// TIA Portal V16 export
// export: Created 2023-03-29T11:03:44.8927615Z, ExportSetting WithDefaults, DisplayName Totally Integrated Automation Portal, DisplayVersion V16 Update 6, DisplayName TIA Portal Version Control Interface, DisplayVersion V16 Update 2, DisplayName TIA Portal Openness, DisplayVersion V16 Update 6, DisplayName STEP 7 Professional, DisplayVersion V16 Update 6, DisplayName STEP 7 Safety, DisplayVersion V16, DisplayName WinCC Advanced, DisplayVersion V16 Update 6
VAR_GLOBAL   // PLC tag table "Z3"
   Hbit_Alarm_Z3 AT %M14.0 : Bool;
   CMD_Open_Z_3 AT %M57.5 : Bool;   // załącz otwieranie
   Hbit_Reset_Z3 AT %M14.6 : Bool;
   CMD_Awaria_Z_3 AT %M57.7 : Bool;   // Awaria zbiorcza
   inputOtwartaZ_3 AT %M56.2 : Bool;   // znacznik wejście
   setAlarm_Moment_Z_3 AT %M57.4 : Bool;   // znacznik alarmu od momentówki w trybie zdalnym (aut/mamnual)
   inputRuch_Z_3 AT %M56.4 : Bool;
   setSVMO_Z_3 AT %M57.2 : Bool;   // Znacznik polecenia otwórz w trybie automat
   CMD_Close_Z_3 AT %M57.6 : Bool;   // załącz zamykanie
   Byte_Status_Z3 AT %MW14 : Word;   // Słowo statusu napędu
   isAUMA_Z_3 AT %M52.4 : Bool;   // przęłącznik wymiany na AUMA
   inputAumagotowośćZ_3 AT %M57.0 : Bool;   // znacznik wejście
   Hbit_Auto_Manu_Z3 AT %M14.7 : Bool;
   inputAumalokalneZ_3 AT %M56.6 : Bool;   // znacznik wejście
   Hbit_Zamknieta_Z3 AT %M14.3 : Bool;
   setSVMC_Z_3 AT %M57.3 : Bool;   // Znacznik polecenia zamknij w trybie automat
   Hbit_REN_Z3 AT %M14.2 : Bool;
   Hbit_Otwórz_Z3 AT %M14.4 : Bool;
   inputAumaawariaZ_3 AT %M57.1 : Bool;   // znacznik wejście
   inputAumaautomatZ_3 AT %M56.7 : Bool;   // znacznik wejście
   inputREMT_Z_3 AT %M56.1 : Bool;   // znacznik wejście zdalne
   inputAwariaMomentZ_3 AT %M56.5 : Bool;   // znacznik wejście
   isGotowość_Z_3 AT %M56.0 : Bool;   // bit gotowości wspólny
   Hbit_Otwarta_Z3 AT %M14.1 : Bool;
   inputZamkniętaZ_3 AT %M56.3 : Bool;   // znacznik wejście
   Hbit_Zamknij_Z3 AT %M14.5 : Bool;
END_VAR
